TYPE ENCControlChannel :
STRUCT
	{attribute addProperty Name "Control"}
	Control AT %Q* : stENCControlCompact;
	{attribute addProperty Name "Set counter value"}
	SetCounterValue AT %Q* : UDINT;
END_STRUCT
END_TYPE

(* stored: Version 1.1.0.1, ProductVersion 3.1.4024.9
   DUT ENCControlChannel: Id {50cd8acc-0c9f-0369-0d14-c0300fecb36c} *)
